FUNCTION_BLOCK FB_AnalogScaling IMPLEMENTS I_AnalogScaling
VAR_INPUT
END_VAR
VAR_OUTPUT
END_VAR
VAR
		fbScaling		: FB_Scaling;
END_VAR

;

METHOD ActualSpeed : REAL
VAR_INPUT
	nRawSensorValue		: REAL;
	nLowerScaleValue	: REAL;
	nHigherScaleValue	: REAL;
	nOutputLowerLimit	: REAL;
	nOutPutHigherLimit	: REAL;
END_VAR
THIS^.fbScaling(
	nRawInputValue		:= nRawSensorValue, 
	nInputLowerLimit	:= nLowerScaleValue , 
	nInputHigherLimit	:= nHigherScaleValue, 
	nOutputLowerLimit	:= nOutputLowerLimit, 
	nOutputHigherLimit	:= nOutPutHigherLimit , 
	nScaledValueF		=> ActualSpeed, 
	nScaledValueD		=> );
END_METHOD

METHOD LoadCell : REAL
VAR_INPUT
	nRawSensorValue		: REAL;
	nLowerScaleValue	: REAL;
	nHigherScaleValue	: REAL;
	nOutputLowerLimit	: REAL;
	nOutPutHigherLimit	: REAL;
END_VAR
THIS^.fbScaling(
	nRawInputValue		:= nRawSensorValue, 
	nInputLowerLimit	:= nLowerScaleValue , 
	nInputHigherLimit	:= nHigherScaleValue, 
	nOutputLowerLimit	:= nOutputLowerLimit, 
	nOutputHigherLimit	:= nOutPutHigherLimit , 
	nScaledValueF		=> LoadCell, 
	nScaledValueD		=> );
END_METHOD

METHOD pH : REAL
VAR_INPUT
	nRawSensorValue		: REAL;
	nLowerScaleValue	: REAL;
	nHigherScaleValue	: REAL;
	nOutputLowerLimit	: REAL;
	nOutPutHigherLimit	: REAL;
END_VAR
THIS^.fbScaling(
	nRawInputValue		:= nRawSensorValue, 
	nInputLowerLimit	:= nLowerScaleValue , 
	nInputHigherLimit	:= nHigherScaleValue, 
	nOutputLowerLimit	:= nOutputLowerLimit, 
	nOutputHigherLimit	:= nOutPutHigherLimit , 
	nScaledValueF		=> pH, 
	nScaledValueD		=> );
END_METHOD

METHOD Pressure : REAL
VAR_INPUT
	nRawSensorValue		: REAL;
	nLowerScaleValue	: REAL;
	nHigherScaleValue	: REAL;
	nOutputLowerLimit	: REAL;
	nOutPutHigherLimit	: REAL;
END_VAR
THIS^.fbScaling(
	nRawInputValue		:= nRawSensorValue, 
	nInputLowerLimit	:= nLowerScaleValue , 
	nInputHigherLimit	:= nHigherScaleValue, 
	nOutputLowerLimit	:= nOutputLowerLimit, 
	nOutputHigherLimit	:= nOutPutHigherLimit , 
	nScaledValueF		=> Pressure, 
	nScaledValueD		=> );
END_METHOD

METHOD Temperature : REAL
VAR_INPUT
	nRawSensorValue		: REAL;
	nLowerScaleValue	: REAL;
	nHigherScaleValue	: REAL;
	nOutputLowerLimit	: REAL;
	nOutPutHigherLimit	: REAL;
END_VAR
THIS^.fbScaling(
	nRawInputValue		:= nRawSensorValue, 
	nInputLowerLimit	:= nLowerScaleValue , 
	nInputHigherLimit	:= nHigherScaleValue, 
	nOutputLowerLimit	:= nOutputLowerLimit, 
	nOutputHigherLimit	:= nOutPutHigherLimit , 
	nScaledValueF		=> Temperature, 
	nScaledValueD		=> );
END_METHOD

END_FUNCTION_BLOCK

(* stored: Version 1.1.0.1, ProductVersion 3.1.4024.4
   POU FB_AnalogScaling: Id {67b6dfba-7acc-4f95-b088-c186f8d756cf}, SpecialFunc None
   Method ActualSpeed: Id {5af5cef2-56a5-40ff-a57a-b73536e7c21c}
   Method LoadCell: Id {f927ed0f-40b1-4a7b-947a-ac888493d410}
   Method pH: Id {91843410-60b2-47ca-adda-27339196593f}
   Method Pressure: Id {9aaafd3b-fd31-46a5-93d6-a4e94da00f15}
   Method Temperature: Id {63386ee9-c744-4e3c-b0ab-b44875ea241b} *)
